FUNCTION_BLOCK Robot_Task_Core (* Basic Function Block Type *)
  (* Standard: 61499-2 *)
  (* Version 0.0, 8/21/2025, Evans_A, Schneider Electric, Template *)
  PACKAGE Main;
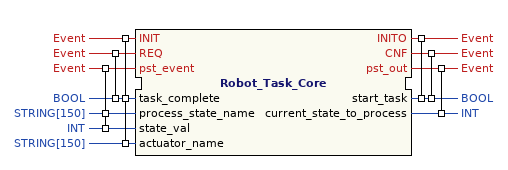
  EVENT_INPUT
    INIT WITH task_complete, actuator_name; (* Initialization Request *)
    REQ WITH task_complete; (* Normal Execution Request *)
    pst_event WITH process_state_name, state_val;
  END_EVENT
  EVENT_OUTPUT
    INITO WITH start_task; (* Initialization Confirm *)
    CNF WITH start_task; (* Execution Confirmation *)
    pst_out WITH current_state_to_process;
  END_EVENT
  VAR_INPUT
    task_complete : BOOL; (* Input event qualifier *)
    process_state_name : STRING[150];
    state_val : INT;
    actuator_name : STRING[150];
  END_VAR
  VAR_OUTPUT
    start_task : BOOL; (* Output event qualifier *)
    current_state_to_process : INT;
  END_VAR
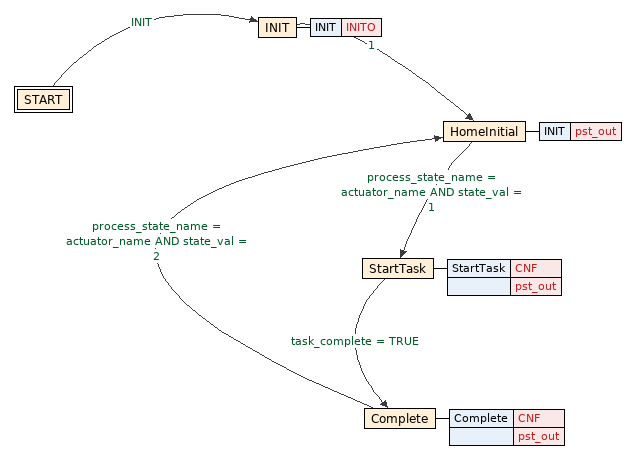
  EC_STATES
    START; (* Initial State *)
    INIT : INIT -> INITO; (* Initialization *)
    StartTask : StartTask -> CNF, -> pst_out; (* Normal execution *)
    Complete : Complete -> CNF, -> pst_out;
    HomeInitial : INIT -> pst_out;
  END_STATES
  EC_TRANSITIONS
    START TO INIT := INIT;
    INIT TO HomeInitial := 1;
    HomeInitial TO StartTask := process_state_name = actuator_name AND state_val = 1;
    StartTask TO Complete := task_complete = TRUE;
    Complete TO HomeInitial := process_state_name = actuator_name AND state_val = 2;
  END_TRANSITIONS
  ALGORITHM INIT IN ST: (* Initialization algorithm *)
start_task := FALSE;
current_state_to_process := 0;
  END_ALGORITHM
  ALGORITHM REQ IN ST: (* Normally executed algorithm *)
;
  END_ALGORITHM
  ALGORITHM StartTask IN ST:
start_task := TRUE;
current_state_to_process := 1;
  END_ALGORITHM
  ALGORITHM Complete IN ST:
start_task := FALSE;
current_state_to_process := 2;
  END_ALGORITHM
END_FUNCTION_BLOCK
